// LS Electric XG5000 project: 0122 PLC 데이터1
// PLC LSPLC

PROGRAM NewProgram (task: 스캔 프로그램)

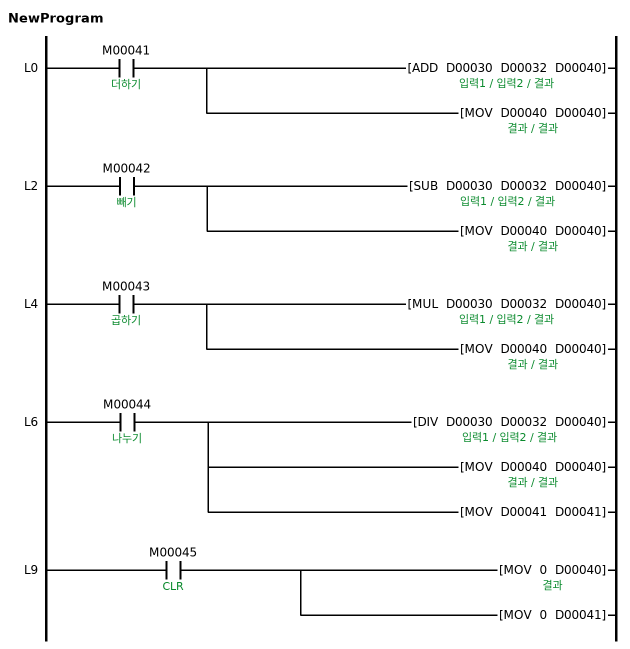
; L0
LOAD      M00041	// 더하기
ADD       D00030 D00032 D00040	// 입력1 / 입력2 / 결과
MOV       D00040 D00040	// 결과 / 결과
; L2
LOAD      M00042	// 빼기
SUB       D00030 D00032 D00040	// 입력1 / 입력2 / 결과
MOV       D00040 D00040	// 결과 / 결과
; L4
LOAD      M00043	// 곱하기
MUL       D00030 D00032 D00040	// 입력1 / 입력2 / 결과
MOV       D00040 D00040	// 결과 / 결과
; L6
LOAD      M00044	// 나누기
DIV       D00030 D00032 D00040	// 입력1 / 입력2 / 결과
MOV       D00040 D00040	// 결과 / 결과
MOV       D00041 D00041
; L9
LOAD      M00045	// CLR
MOV       0 D00040	// 결과
MOV       0 D00041

VARIABLES AND COMMENTS (devices not used above)
M00010	BIT	스위치 1
D00000	WORD	전번
M00001	BIT	스위치2
D00022	WORD	현재카운터수
M00002	BIT	스위치3
M00003	BIT	카운터
M00004	BIT	카운터 리셋
C0000	BIT/WORD	카운트
M00000	BIT	스위치1